TYPE ST_OutputsLoadstacker :
STRUCT
	HW					: ST_HW_OutputLoadStacker;		
END_STRUCT
END_TYPE

(* stored: Version 1.1.0.1, ProductVersion 3.1.4024.4
   DUT ST_OutputsLoadstacker: Id {ad6e3966-047f-4a98-b351-145c0f79ef16} *)
